FUNCTION_BLOCK FB_Conveyor
VAR_INPUT
	
END_VAR
VAR_OUTPUT
END_VAR
VAR
	Timer1 : Tc2_Standard.TON;
	Step_0_Standby : BOOL;
	Step_0: BOOL;
	Step_1 : BOOL;
	Step_2 : BOOL;
	Step_3 : BOOL;
	Step_4 : BOOL;
	Step_5 : BOOL;
	Step_6 : BOOL;
	
END_VAR
VAR_IN_OUT
	control_data : Plant_CTRL;
	control_data_vision : CM_Vision_UDT;
	control_data_Conveyor1 : CM_DO_UDT;
	
	control_data_StopBlade : CM_DO_UDT;
	control_data_emitter : CM_DO_UDT;
END_VAR
VAR // added by the converter: edge detectors and wires of the graphical bodies
    _w1, _w2, _w3, _w4, _w5, _w6, _w7, _w8, _w9, _w10 : BOOL;
END_VAR

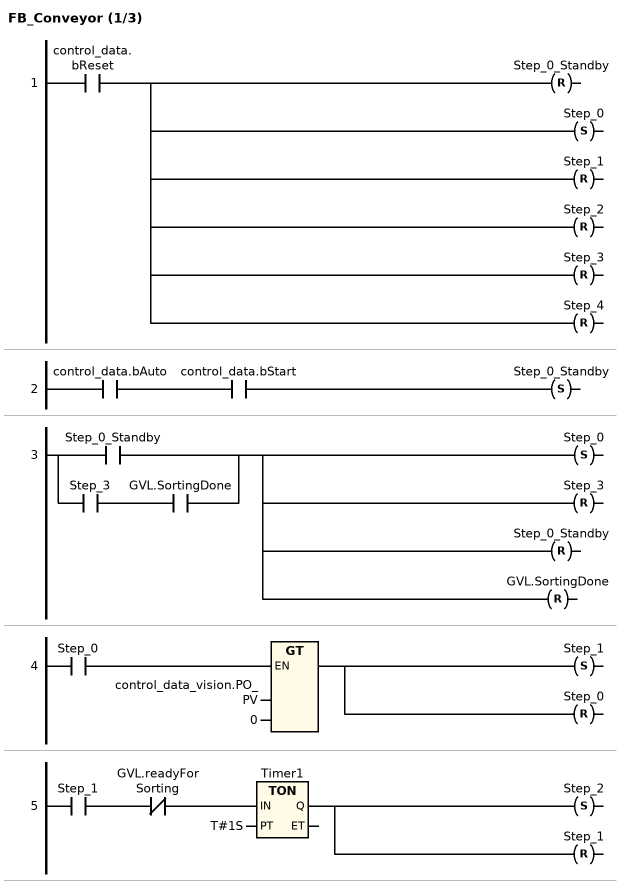
// NETWORK 1
Step_0_Standby R= control_data.bReset;
Step_0 S= control_data.bReset;
Step_1 R= control_data.bReset;
Step_2 R= control_data.bReset;
Step_3 R= control_data.bReset;
Step_4 R= control_data.bReset;

// NETWORK 2
Step_0_Standby S= control_data.bAuto AND control_data.bStart;

// NETWORK 3
_w1 := Step_0_Standby OR Step_3 AND GVL.SortingDone;
Step_0 S= _w1;
Step_3 R= _w1;
Step_0_Standby R= _w1;
GVL.SortingDone R= _w1;

// NETWORK 4
_w2 := Step_0 AND control_data_vision.PO_PV > 0;
Step_1 S= _w2;
Step_0 R= _w2;

// NETWORK 5
Timer1(IN := Step_1 AND NOT GVL.readyForSorting, PT := T#1S); // TON
Step_2 S= Timer1.Q;
Step_1 R= Timer1.Q;

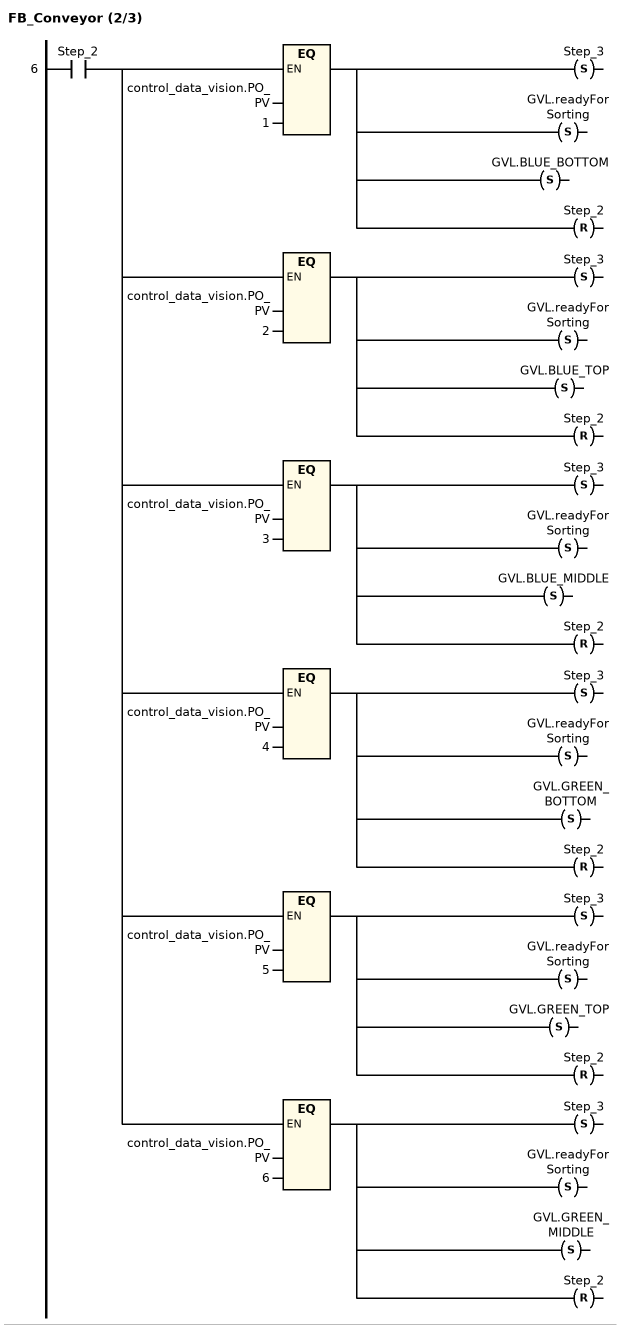
// NETWORK 6
_w3 := Step_2;
_w4 := _w3 AND control_data_vision.PO_PV = 1;
Step_3 S= _w4;
GVL.readyForSorting S= _w4;
GVL.BLUE_BOTTOM S= _w4;
Step_2 R= _w4;
_w5 := _w3 AND control_data_vision.PO_PV = 2;
Step_3 S= _w5;
GVL.readyForSorting S= _w5;
GVL.BLUE_TOP S= _w5;
Step_2 R= _w5;
_w6 := _w3 AND control_data_vision.PO_PV = 3;
Step_3 S= _w6;
GVL.readyForSorting S= _w6;
GVL.BLUE_MIDDLE S= _w6;
Step_2 R= _w6;
_w7 := _w3 AND control_data_vision.PO_PV = 4;
Step_3 S= _w7;
GVL.readyForSorting S= _w7;
GVL.GREEN_BOTTOM S= _w7;
Step_2 R= _w7;
_w8 := _w3 AND control_data_vision.PO_PV = 5;
Step_3 S= _w8;
GVL.readyForSorting S= _w8;
GVL.GREEN_TOP S= _w8;
Step_2 R= _w8;
_w9 := _w3 AND control_data_vision.PO_PV = 6;
Step_3 S= _w9;
GVL.readyForSorting S= _w9;
GVL.GREEN_MIDDLE S= _w9;
Step_2 R= _w9;

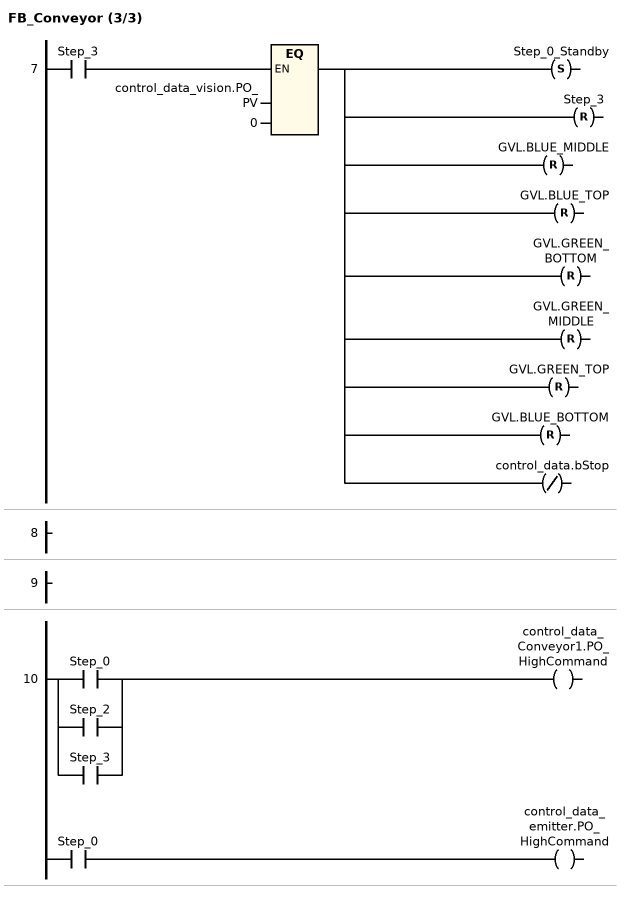
// NETWORK 7
_w10 := Step_3 AND control_data_vision.PO_PV = 0;
Step_0_Standby S= _w10;
Step_3 R= _w10;
GVL.BLUE_MIDDLE R= _w10;
GVL.BLUE_TOP R= _w10;
GVL.GREEN_BOTTOM R= _w10;
GVL.GREEN_MIDDLE R= _w10;
GVL.GREEN_TOP R= _w10;
GVL.BLUE_BOTTOM R= _w10;
control_data.bStop := NOT _w10;

// NETWORK 8

// NETWORK 9

// NETWORK 10
control_data_Conveyor1.PO_HighCommand := Step_0 OR Step_2 OR Step_3;
control_data_emitter.PO_HighCommand := Step_0;

END_FUNCTION_BLOCK

(* stored: Version 1.1.0.1, ProductVersion 3.1.4024.13
   POU FB_Conveyor: Id {0cbf57b1-20ed-4dcc-924e-31c53c86553a}, SpecialFunc None *)
